FUNCTION_BLOCK PUBLIC FB_RS_TRIG
VAR_INPUT
	CLK : BOOL;
END_VAR
VAR_OUTPUT
	Q : BOOL; // pos edge
	QS : BOOL; // pos edge set
END_VAR
VAR
	Trig : R_TRIG;
END_VAR

Trig(CLK := CLK, Q => Q);
IF Trig.Q THEN
	QS := TRUE;
END_IF;

METHOD PUBLIC Reset : REFERENCE TO FB_RS_TRIG
VAR_INPUT
END_VAR
THIS^.QS := FALSE;

Reset REF= THIS^;
END_METHOD

END_FUNCTION_BLOCK

(* stored: Version 1.1.0.1, ProductVersion 3.1.4024.12
   POU FB_RS_TRIG: Id {5e76f356-e397-4f73-853a-f86f47d47ef4}, SpecialFunc None
   Method Reset: Id {e4f6ffeb-289d-4606-9e9e-9a4a9ddc8329} *)
